Fanuc KAREL source: NC0050.KL

-- PROVISIONAL review KL for V940-1; original PC SHA256 a60c87f8798f84a1b256da544913f2d22b5702e7dcd2efc2a71bcbfe310bdd7b
-- Incomplete behavior may be omitted. Consult companion uncertainty JSON. Do not deploy.
PROGRAM NC0050
%NOLOCKGROUP
-- UNRESOLVED_LOCAL_POOL 1 cells at code offset 3; source declarations unknown
-- DIRECT_LOCAL_WORD_ACCESS alone does not prove INTEGER, REAL, or BOOLEAN
BEGIN
  -- V9_CONDITION_STACK_HINT 9 bounded expression windows; static native code-base-relative target link; source arms held
  -- UNRESOLVED_PC offsets 0-8; opcodes 2B,2C,7B
  -- UNRESOLVED_PC offsets 13-20; opcodes 9D,23
  -- UNRESOLVED_PC offsets 25-38; opcodes 21,9D,57,79
  -- UNRESOLVED_PC offsets 43-60; opcodes 21,40,41,42
  -- UNRESOLVED_PC offsets 65-78; opcodes 21,9D,57,79
  -- UNRESOLVED_PC offsets 83-100; opcodes 21,40,41,42
  -- UNRESOLVED_PC offsets 105-118; opcodes 21,9D,57,79
  -- UNRESOLVED_PC offsets 123-140; opcodes 21,40,41,42
  -- UNRESOLVED_PC offsets 145-158; opcodes 21,9D,57,79
  -- UNRESOLVED_PC offsets 163-180; opcodes 21,40,41,42
  -- UNRESOLVED_PC offsets 185-198; opcodes 21,9D,57,79
  -- UNRESOLVED_PC offsets 203-220; opcodes 21,40,41,42
  -- UNRESOLVED_PC offsets 225-238; opcodes 21,9D,57,79
  -- UNRESOLVED_PC offsets 243-260; opcodes 21,40,41,42
  -- UNRESOLVED_PC offsets 265-278; opcodes 21,9D,57,79
  -- UNRESOLVED_PC offsets 283-300; opcodes 21,40,41,42
  -- UNRESOLVED_PC offsets 305-318; opcodes 21,9D,57,79
  -- UNRESOLVED_PC offsets 323-340; opcodes 21,40,41,42
  -- UNRESOLVED_PC offsets 345-358; opcodes 21,9D,57,79
  -- UNRESOLVED_PC offsets 363-380; opcodes 21,40,41,42
  -- UNRESOLVED_PC offsets 385-415; opcodes 21,9D,52,23,7A,40,41,42
  -- UNRESOLVED_PC offsets 420-444; opcodes 21,2E,52,23,7A,43
  -- UNRESOLVED_PC offsets 449-467; opcodes 21,2E,52,23
  -- UNRESOLVED_PC offsets 477-482; opcodes 7A
  -- UNRESOLVED_PC offsets 487-505; opcodes 21,2E,52,23
  -- UNRESOLVED_PC offsets 510-526; opcodes 7A,40,41,42
  -- UNRESOLVED_PC offsets 531-555; opcodes 21,2E,52,23,7A,43
  -- UNRESOLVED_PC offsets 560-578; opcodes 21,2E,52,23
  -- UNRESOLVED_PC offsets 588-593; opcodes 7A
  -- UNRESOLVED_PC offsets 598-616; opcodes 21,2E,52,23
  -- UNRESOLVED_PC offsets 621-637; opcodes 7A,40,41,42
  -- UNRESOLVED_PC offsets 642-666; opcodes 21,2E,52,23,7A,43
  -- UNRESOLVED_PC offsets 671-689; opcodes 21,2E,52,23
  -- UNRESOLVED_PC offsets 699-704; opcodes 7A
  -- UNRESOLVED_PC offsets 709-727; opcodes 21,2E,52,23
  -- UNRESOLVED_PC offsets 732-748; opcodes 7A,40,41,42
  -- UNRESOLVED_PC offsets 753-777; opcodes 21,2E,52,23,7A,43
  -- UNRESOLVED_PC offsets 782-800; opcodes 21,2E,52,23
  -- UNRESOLVED_PC offsets 810-815; opcodes 7A
  -- UNRESOLVED_PC offsets 820-838; opcodes 21,2E,52,23
  -- UNRESOLVED_PC offsets 843-859; opcodes 7A,40,41,42
  -- UNRESOLVED_PC offsets 864-888; opcodes 21,2E,52,23,7A,43
  -- UNRESOLVED_PC offsets 893-911; opcodes 21,2E,52,23
  -- UNRESOLVED_PC offsets 921-926; opcodes 7A
  -- UNRESOLVED_PC offsets 931-949; opcodes 21,2E,52,23
  -- UNRESOLVED_PC offsets 954-970; opcodes 7A,40,41,42
  -- UNRESOLVED_PC offsets 975-999; opcodes 21,2E,52,23,7A,43
  -- UNRESOLVED_PC offsets 1004-1022; opcodes 21,2E,52,23
  -- UNRESOLVED_PC offsets 1032-1037; opcodes 7A
  -- UNRESOLVED_PC offsets 1042-1060; opcodes 21,2E,52,23
  -- UNRESOLVED_PC offsets 1065-1081; opcodes 7A,40,41,42
  -- UNRESOLVED_PC offsets 1086-1110; opcodes 21,2E,52,23,7A,43
  -- UNRESOLVED_PC offsets 1115-1133; opcodes 21,2E,52,23
  -- UNRESOLVED_PC offsets 1143-1148; opcodes 7A
  -- UNRESOLVED_PC offsets 1153-1171; opcodes 21,2E,52,23
  -- UNRESOLVED_PC offsets 1176-1192; opcodes 7A,40,41,42
  -- UNRESOLVED_PC offsets 1197-1221; opcodes 21,2E,52,23,7A,43
  -- UNRESOLVED_PC offsets 1226-1244; opcodes 21,2E,52,23
  -- UNRESOLVED_PC offsets 1254-1259; opcodes 7A
  -- UNRESOLVED_PC offsets 1264-1282; opcodes 21,2E,52,23
  -- UNRESOLVED_PC offsets 1287-1303; opcodes 7A,40,41,42
  -- UNRESOLVED_PC offsets 1308-1332; opcodes 21,2E,52,23,7A,43
  -- UNRESOLVED_PC offsets 1337-1355; opcodes 21,2E,52,23
  -- UNRESOLVED_PC offsets 1365-1370; opcodes 7A
  -- UNRESOLVED_PC offsets 1375-1393; opcodes 21,2E,52,23
  -- UNRESOLVED_PC offsets 1403-1407; opcodes 7F
  -- UNRESOLVED_PC offsets 1412-1416; opcodes 27,AA
  -- UNRESOLVED_PC offsets 1421-1425; opcodes 7F
END NC0050
